SYSTEM Smart_Grid_02
  (* Version 1.0, 2021-02-16, badger *)
  APPLICATION Smart_Grid_02App
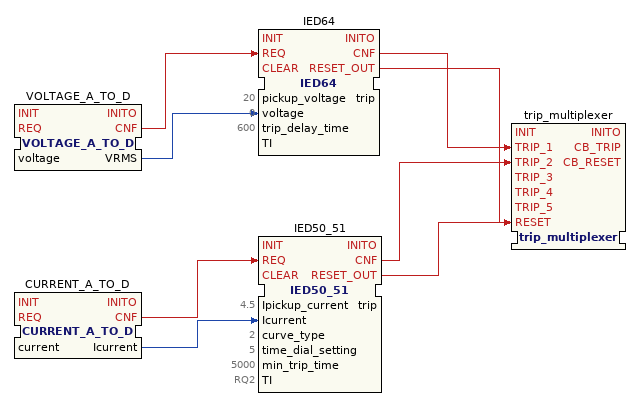
    FBS
      trip_multiplexer : trip_multiplexer;
      IED50_51 : IED50_51(Ipickup_current := 4.5, curve_type := 2, time_dial_setting := 5, min_trip_time := 5000, TI := RQ2);
      IED64 : IED64(pickup_voltage := 20, voltage := 0, trip_delay_time := 600);
      VOLTAGE_A_TO_D : VOLTAGE_A_TO_D;
      CURRENT_A_TO_D : CURRENT_A_TO_D;
    END_FBS
    EVENT_CONNECTIONS
      IED50_51.CNF TO trip_multiplexer.TRIP_2;
      IED50_51.RESET_OUT TO trip_multiplexer.RESET;
      IED64.CNF TO trip_multiplexer.TRIP_1;
      IED64.RESET_OUT TO trip_multiplexer.RESET;
      VOLTAGE_A_TO_D.CNF TO IED64.REQ;
      CURRENT_A_TO_D.CNF TO IED50_51.REQ;
    END_CONNECTIONS
    DATA_CONNECTIONS
      VOLTAGE_A_TO_D.VRMS TO IED64.voltage;
      CURRENT_A_TO_D.Icurrent TO IED50_51.Icurrent;
    END_CONNECTIONS
  END_APPLICATION
  DEVICE FORTE_PC_1 : FORTE_PC(MGR_ID := "localhost:61499")
    {SET_ATTRIBUTE(Profile, HOLOBLOC)} (* device profile *)
    RESOURCE SMART_GRID : EMB_RES
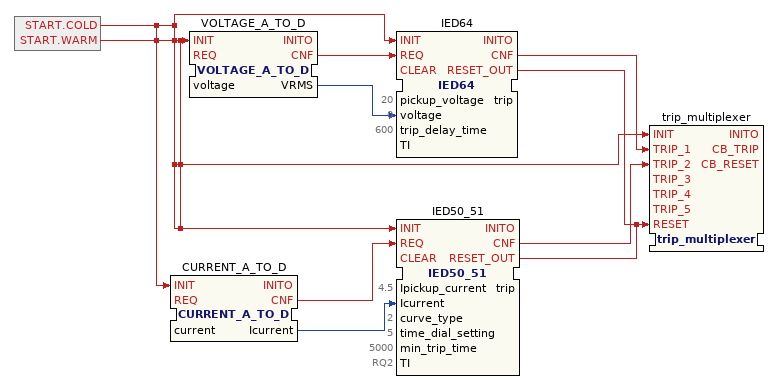
      FBS
        trip_multiplexer : trip_multiplexer;
        IED50_51 : IED50_51(Ipickup_current := 4.5, curve_type := 2, time_dial_setting := 5, min_trip_time := 5000, TI := RQ2);
        IED64 : IED64(pickup_voltage := 20, voltage := 0, trip_delay_time := 600);
        VOLTAGE_A_TO_D : VOLTAGE_A_TO_D;
        CURRENT_A_TO_D : CURRENT_A_TO_D;
      END_FBS
      EVENT_CONNECTIONS
        START.COLD TO trip_multiplexer.INIT;
        START.WARM TO trip_multiplexer.INIT;
        IED50_51.CNF TO trip_multiplexer.TRIP_2;
        IED50_51.RESET_OUT TO trip_multiplexer.RESET;
        IED64.CNF TO trip_multiplexer.TRIP_1;
        IED64.RESET_OUT TO trip_multiplexer.RESET;
        START.COLD TO IED64.INIT;
        START.WARM TO IED64.INIT;
        START.COLD TO IED50_51.INIT;
        START.WARM TO IED50_51.INIT;
        VOLTAGE_A_TO_D.CNF TO IED64.REQ;
        CURRENT_A_TO_D.CNF TO IED50_51.REQ;
        START.COLD TO VOLTAGE_A_TO_D.INIT;
        START.COLD TO CURRENT_A_TO_D.INIT;
        START.WARM TO CURRENT_A_TO_D.INIT;
      END_CONNECTIONS
      DATA_CONNECTIONS
        VOLTAGE_A_TO_D.VRMS TO IED64.voltage;
        CURRENT_A_TO_D.Icurrent TO IED50_51.Icurrent;
      END_CONNECTIONS
    END_RESOURCE
  END_DEVICE
  MAPPINGS
    Smart_Grid_02App.trip_multiplexer ON FORTE_PC_1.SMART_GRID.trip_multiplexer;
    Smart_Grid_02App.IED50_51 ON FORTE_PC_1.SMART_GRID.IED50_51;
    Smart_Grid_02App.IED64 ON FORTE_PC_1.SMART_GRID.IED64;
    Smart_Grid_02App.VOLTAGE_A_TO_D ON FORTE_PC_1.SMART_GRID.VOLTAGE_A_TO_D;
    Smart_Grid_02App.CURRENT_A_TO_D ON FORTE_PC_1.SMART_GRID.CURRENT_A_TO_D;
  END_MAPPINGS
  SEGMENTS
    Ethernet : Ethernet;
  END_SEGMENTS
  LINKS
    FORTE_PC_1 => Ethernet;
  END_LINKS
END_SYSTEM
